// TIA Portal V15.1 export
// export: Created 2024-06-21T08:41:10.3713912Z, ExportSetting WithDefaults, DisplayName Totally Integrated Automation Portal, DisplayVersion V15.1 Update 5, DisplayName TIA Portal Openness, DisplayVersion V15.1 Update 5, DisplayName SINAMICS Startdrive Advanced, DisplayVersion V15.1, DisplayName G130, G150, S120, S150, SINAMICS MV, S210, DisplayVersion V15.1, DisplayName G110M, G120, G120C, G120D, G120P, DisplayVersion V15.1, DisplayName STEP 7 Professional, DisplayVersion V15.1 Update 5, DisplayName STEP 7 Safety, DisplayVersion V15.1, DisplayName WinCC Professional, DisplayVersion V15.1 Update 5, DisplayName SIMATIC Visualization Architect, DisplayVersion V15.1
FUNCTION "LGBLineConv-MDXPN-Config" : Void   // FC6640, FBD
TITLE = LCrossConv2W2S-G120PN-Config / LGBLineConvMDXPN-Config
{ S7_Optimized_Access := 'FALSE' }
AUTHOR : VCC
FAMILY : Config
NAME : Bit2Word
VERSION : 0.1
// =============================================================================
// Handles the LCross2W2SG120PN Config
// =============================================================================
// stored: AutoNumber false, IsIECCheckEnabled false, SetENOAutomatically False, UDAEnableTagReadback false
   VAR_INPUT
      C_DetMinGapLeftUsed : Bool;   // Input 0 / Config / Lowspeed stop detection Set used
      C_DetMinGapRightUsed : Bool;   // Input 0 / Config / Lowspeed stop detection Set used
      C_BothDetMinGapIsAlarmB : Bool;   // Config
      C_OneDetMinGapIsAlarmC : Bool;   // Config
      C_InitDirection : Bool;   // Input 7 / Config
      C_SafetySwNc : Bool;   // Input 15 / Config
      C_SafetySwUsed : Bool;   // Input 16 / Config
      C_MotorProtectionNc : Bool;   // Motorprotection NC / Config
      C_MotorProtectionUsed : Bool;   // Motorprotection NC / Config
      C_BrakeProtectionNc : Bool;   // Config
      C_BrakeProtectionUsed : Bool;   // Config
      C_MotionStopUsed : Bool;   // Config
      C_EnableAlarmHW : Bool;   // Enable Alarm hardware (e.g. safetyswitch, motorprotector, detections) / Enable Alarm hardware (e.g. Safetyswitch, Motorprotector, detections) / Config
      C_EnableAlarmTransfer : Bool;   // Enable Alarm transfer (e.g. Transfer in , transfer out) / Config
      C_DetSaturationDelay : Time;   // Config
      C_Ramp : Time;   // Config
      C_ReferenceDriveCurrent : Real;   // Config
      C_ReferenceMotorCurrent : Real;   // Config
      C_ReferenceMotorRPM : Real;   // Config
      C_RatioGearbox : Real;   // Config
      C_Diameter : Real;   // Config
      C_Acceleration : Real;   // Config
      C_TrfMaxTime : DInt;   // Max allowed transfertime (millisec) / Config
      C_AllowedResetDirection : Bool;   // Config
      C_MaxTimeResetDirection : DInt;   // Config
      C_AllowedEcoMode : Bool;   // Config
      C_TimeEcoMode : Time;   // Config
      C_HWSubInput : HW_SUBMODULE;   // I/O / Config
      C_HWSubOutput : HW_SUBMODULE;   // I/O / Config
   END_VAR
   VAR_IN_OUT
      IO_Config : "LineConv-MDXPNConfig";   // Config
   END_VAR
BEGIN

REGION Network 1: **** 1 - Inputs **** Move Config
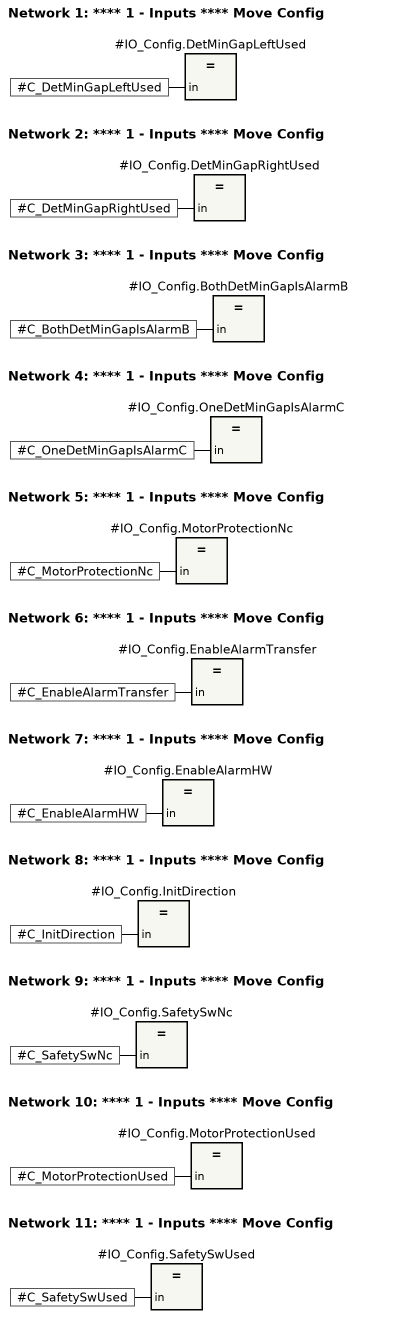
   #IO_Config.DetMinGapLeftUsed := #C_DetMinGapLeftUsed;
END_REGION

REGION Network 2: **** 1 - Inputs **** Move Config
   #IO_Config.DetMinGapRightUsed := #C_DetMinGapRightUsed;
END_REGION

REGION Network 3: **** 1 - Inputs **** Move Config
   #IO_Config.BothDetMinGapIsAlarmB := #C_BothDetMinGapIsAlarmB;
END_REGION

REGION Network 4: **** 1 - Inputs **** Move Config
   #IO_Config.OneDetMinGapIsAlarmC := #C_OneDetMinGapIsAlarmC;
END_REGION

REGION Network 5: **** 1 - Inputs **** Move Config
   // Move Config
   #IO_Config.MotorProtectionNc := #C_MotorProtectionNc;
END_REGION

REGION Network 6: **** 1 - Inputs **** Move Config
   // Move Config
   #IO_Config.EnableAlarmTransfer := #C_EnableAlarmTransfer;
END_REGION

REGION Network 7: **** 1 - Inputs **** Move Config
   // Move Config
   #IO_Config.EnableAlarmHW := #C_EnableAlarmHW;
END_REGION

REGION Network 8: **** 1 - Inputs **** Move Config
   // Move Config
   #IO_Config.InitDirection := #C_InitDirection;
END_REGION

REGION Network 9: **** 1 - Inputs **** Move Config
   // Move Config
   #IO_Config.SafetySwNc := #C_SafetySwNc;
END_REGION

REGION Network 10: **** 1 - Inputs **** Move Config
   // Move Config
   #IO_Config.MotorProtectionUsed := #C_MotorProtectionUsed;
END_REGION

REGION Network 11: **** 1 - Inputs **** Move Config
   // Move Config
   #IO_Config.SafetySwUsed := #C_SafetySwUsed;
END_REGION

REGION Network 12: **** 1 - Inputs **** Move Config
   // Move Config
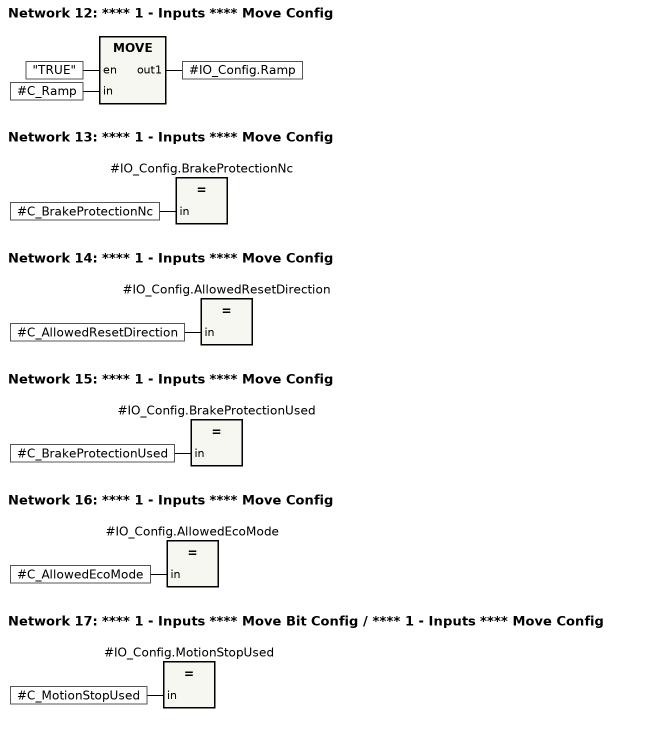
   IF "TRUE" THEN #IO_Config.Ramp := #C_Ramp; END_IF;
END_REGION

REGION Network 13: **** 1 - Inputs **** Move Config
   // Move Config
   #IO_Config.BrakeProtectionNc := #C_BrakeProtectionNc;
END_REGION

REGION Network 14: **** 1 - Inputs **** Move Config
   #IO_Config.AllowedResetDirection := #C_AllowedResetDirection;
END_REGION

REGION Network 15: **** 1 - Inputs **** Move Config
   // Move Config
   #IO_Config.BrakeProtectionUsed := #C_BrakeProtectionUsed;
END_REGION

REGION Network 16: **** 1 - Inputs **** Move Config
   // Move Config
   #IO_Config.AllowedEcoMode := #C_AllowedEcoMode;
END_REGION

REGION Network 17: **** 1 - Inputs **** Move Bit Config / **** 1 - Inputs **** Move Config
   // Move Bit Config / Move Config
   #IO_Config.MotionStopUsed := #C_MotionStopUsed;
END_REGION

NETWORK
TITLE = **** 8 - Outputs **** Move Config UDT
// Move Config
      L     #C_ReferenceMotorCurrent;
      T     #IO_Config.ReferenceMotorCurrent;
      L     #C_ReferenceMotorRPM;
      T     #IO_Config.ReferenceMotorRPM;
      L     #C_RatioGearbox;
      T     #IO_Config.RatioGearbox;
      L     #C_Diameter;
      T     #IO_Config.Diameter;
      L     #C_Acceleration;
      T     #IO_Config.Acceleration;
      L     #C_ReferenceDriveCurrent;
      T     #IO_Config.ReferenceDriveCurrent;
      L     #C_DetSaturationDelay;
      T     #IO_Config.DetSaturationDelay;
      L     #C_TrfMaxTime;
      T     #IO_Config.TrfMaxTime;
      L     #C_MaxTimeResetDirection;
      T     #IO_Config.MaxTimeResetDirection;
      L     #C_TimeEcoMode;
      T     #IO_Config.TimeEcoMode;
      L     #C_HWSubInput;
      T     #IO_Config.HWSubInput;
      L     #C_HWSubOutput;
      T     #IO_Config.HWSubOutput;

END_FUNCTION
